// TIA Portal project "Micromaster4_with_S7_1200" (V14)

(* hardware
DEVICE "S7-1200 station_1"  S7-1200 Station
   slot 0: "Rack_0"  S7-1200 Rack  Rack  V1.0
   slot 1: "PLC_1"  CPU 1214C DC/DC/DC  6ES7 214-1AE30-0XB0  V2.0
   slot 2: "AI 4x13BIT_1"  SM 1231 AI4  6ES7 231-4HD30-0XB0  V1.0
   slot 3: "AI 4x13BIT_2"  SM 1231 AI4  6ES7 231-4HD30-0XB0  V1.0
   slot 4: "AQ 2x14BIT_1"  6ES7 232-4HB30-0XB0  V1.0
   slot 101: "CM 1243-5"  CM 1243-5  6GK7 243-5DX30-0XE0  V1.0
DEVICE "GSD device_1"  GSD.Device
   slot 0: "Rack_0"  Rail
   slot 0: "Slave_1"  6SE640X-1PB00-0AA0  V1.0
*)

// ===== PLC "PLC_1"  CPU 1214C DC/DC/DC =====

VAR_GLOBAL   // PLC tag table "Default tag table"
   "Tag_1" AT %M0.0 : Bool;
   "Ready_mode" AT %M0.1 : Bool;
   "Run" AT %M0.2 : Bool;
   "CCW" AT %M0.3 : Bool;
   "OFF2" AT %M0.4 : Bool;
   "OFF3" AT %M0.5 : Bool;
   "Ack" AT %M0.6 : Bool;
   "Control_wrd_1" AT %MW2 : Word;
   "freq" AT %MD4 : Real;
   "write_comm_err" AT %M0.7 : Bool;
   "write_Drive_err" AT %M1.0 : Bool;
   "sent_Dn_flag" AT %M1.1 : Bool;
   "status_wrd" AT %MW8 : Word;
   "actual_freq" AT %MD10 : Real;
   "receive_comm_err" AT %M1.2 : Bool;
   "recieve_dn_flag" AT %M1.3 : Bool;
   "ready_for_on_status" AT %M1.4 : Bool;
   "ready_for_run_status" AT %M1.5 : Bool;
   "operation_on_status" AT %M1.6 : Bool;
   "fault_on" AT %M1.7 : Bool;
   "starting_LOckout__status" AT %M14.0 : Bool;
   "alarm_on" AT %M14.1 : Bool;
   "Motor_overload" AT %M14.2 : Bool;
   "Drive_overload" AT %M14.3 : Bool;
   "Tag_2" AT %MW50 : Word;
   "dummy_bit" AT %M400.1 : Bool;
   "dummy1" AT %MW400 : Word;
   "dummy2" AT %MW402 : Word;
END_VAR

FUNCTION "Micormaster_Write_Data" : Void   // FC1, FBD
TITLE = Micromaster Data Write
{ S7_Optimized_Access := 'TRUE' }
VERSION : 0.1
// Description: This function is used to send the 2 PZD words.
// Author: Ahmed Abd Alrahiem
// Email: a.abdalrahiem@gmail.com
// Last Modification Date: July 9, 2021
   VAR_INPUT
      Control_Word : Word;   // Contains the control word1 that should be transferred to the drive
      Set_Point : Real;   // The set point to be transferred to drive
      WR_HW_ID : Hw_Io;   // The module ID for the PZD words
      Reference_frequency_P2000 : Int;   // The reference frequemcy written to the P2000 parameter
   END_VAR
   VAR_OUTPUT
      Access_Comm_Error : Bool;   // IF set, there is a problem regarding the connection with the drive
      Drive_Error : Bool;   // IF set, there is a problem in the drive and the drive can send no data
      Done : Bool;   // IF set, there is no problem and the data is already written
   END_VAR
   VAR_TEMP
      To_Inverter : Array[1..2] of Word;
      Normalized_setpoint : Word;
      temp_SP_1 : Real;
      temp_SP_2 : Real;
      error_word : Int;
   END_VAR
BEGIN

REGION Network 1
   // Normalization of the setpoint
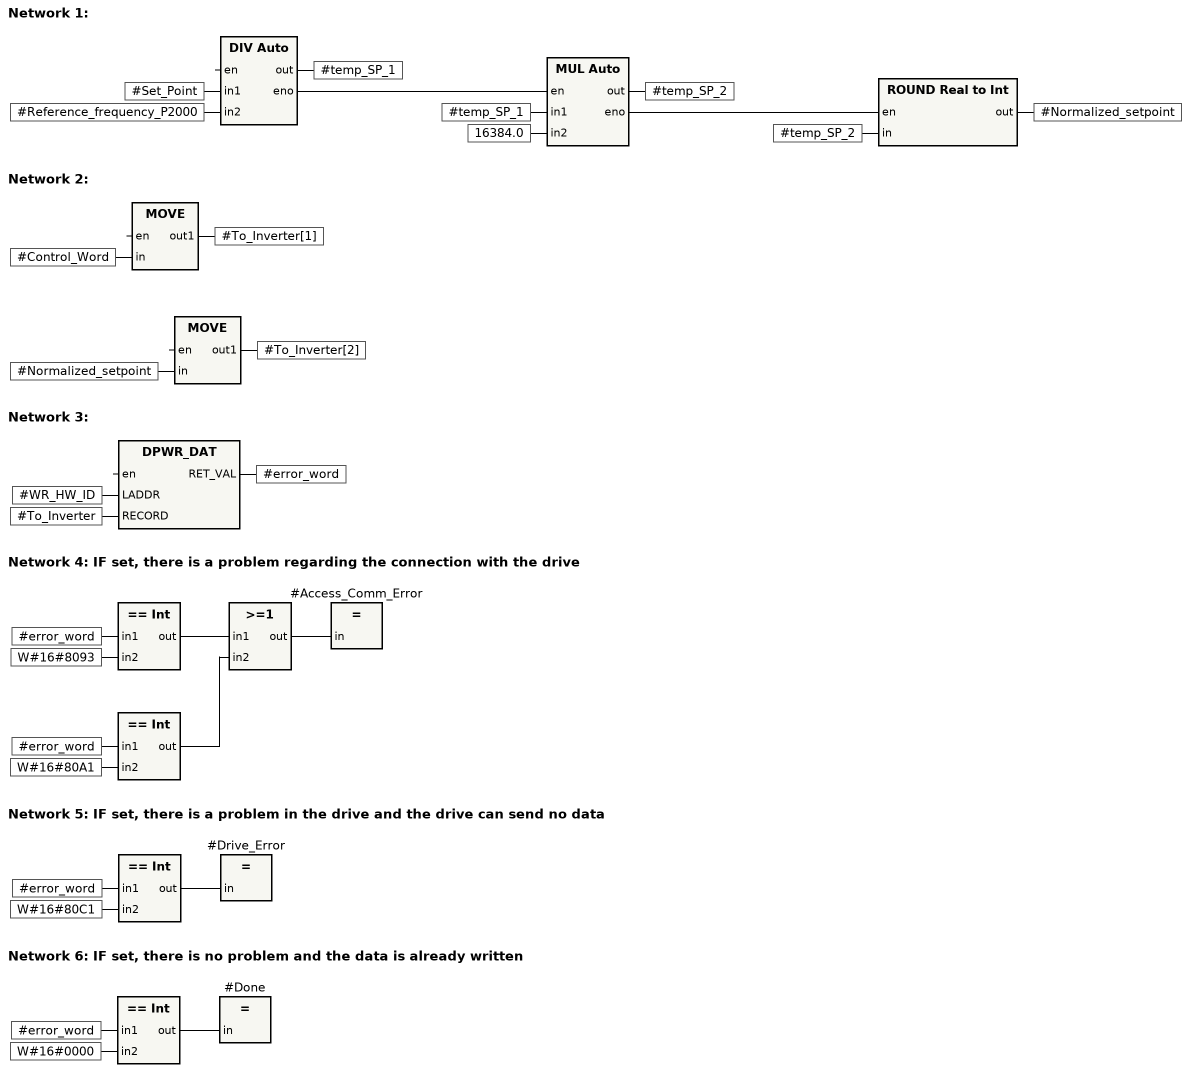
   // ENO of a box is taken as its EN; it also drops when the box reports an error
   #temp_SP_1 := #Set_Point / #Reference_frequency_P2000;
   #temp_SP_2 := #temp_SP_1 * 16384.0;
   #Normalized_setpoint := ROUND(#temp_SP_2);
END_REGION

REGION Network 2
   // This line moves the telegram's control word and setpoint to the same address #To_Inverter
   #To_Inverter[1] := #Control_Word;
   #To_Inverter[2] := #Normalized_setpoint;
END_REGION

REGION Network 3
   // This line writes the data consistently to the inverter
   #error_word := DPWR_DAT(LADDR := #WR_HW_ID, RECORD := #To_Inverter);
END_REGION

REGION Network 4: IF set, there is a problem regarding the connection with the drive
   // The output #Access_Comm_Error is set if there is a problem regarding the connection with the drive
   #Access_Comm_Error := (#error_word = W#16#8093) OR (#error_word = W#16#80A1);
END_REGION

REGION Network 5: IF set, there is a problem in the drive and the drive can send no data
   // The output #Drive_Error is set if there is a problem in the drive and the drive can send no data
   #Drive_Error := #error_word = W#16#80C1;
END_REGION

REGION Network 6: IF set, there is no problem and the data is already written
   // The output #Done is set if there is no problem and the data is already written.
   #Done := #error_word = W#16#0000;
END_REGION
END_FUNCTION

FUNCTION "Micromaster_Control_word1_Generator" : Void   // FC2, FBD
TITLE = Micromaster Control word1 Generator
{ S7_Optimized_Access := 'TRUE' }
VERSION : 0.1
// Description: This function is used to generate the control word to be sent to the Micromaster drive
// Author: Ahmed Abd Alrahiem
// Email: a.abdalrahiem@gmail.com
// Last Modification Date: July 9, 2021
   VAR_INPUT
      "Ready/OFF1" : Bool;   // If set, the inverter will be put in the ready mode--> (bit 0 is set).
      Run : Bool;   // If set, the inverter will be put in the closed loop run mode--> (bit 3 is set).
      CCW_Direction : Bool;   // If set, the motor will run in counter clockwise direction--> (bit 11 is set).
      OFF2 : Bool;   // If set, the drive will coasts to a standstill (Instantaneous braking)-->(bit 1 is reset).
      OFF3 : Bool;   // If set, the drive will shutdown the motor at the fastest possible acceleration rate (rapid shutdown)->(bit 2 is reset).
      Acknowledge_Fault : Bool;   // If set, the inverter fault will be acknowledget--> (bit 7 is set).
   END_VAR
   VAR_OUTPUT
      Control_Word : Word;   // Contains the control word1 that should be transferred to the drive
   END_VAR
   VAR_TEMP
      Control_word_temp1 : Word;
      Control_word_temp2 : Word;
      Control_word_temp3 : Word;
      Control_word_temp4 : Word;
      Control_word_temp5 : Word;
      Control_word_temp6 : Word;
      Control_word_temp7 : Word;
      OFF2_is_reset : Bool;
      OFF3_is_reset : Bool;
   END_VAR
BEGIN

REGION Network 1
   // Moving an initail value equals zero to all bits
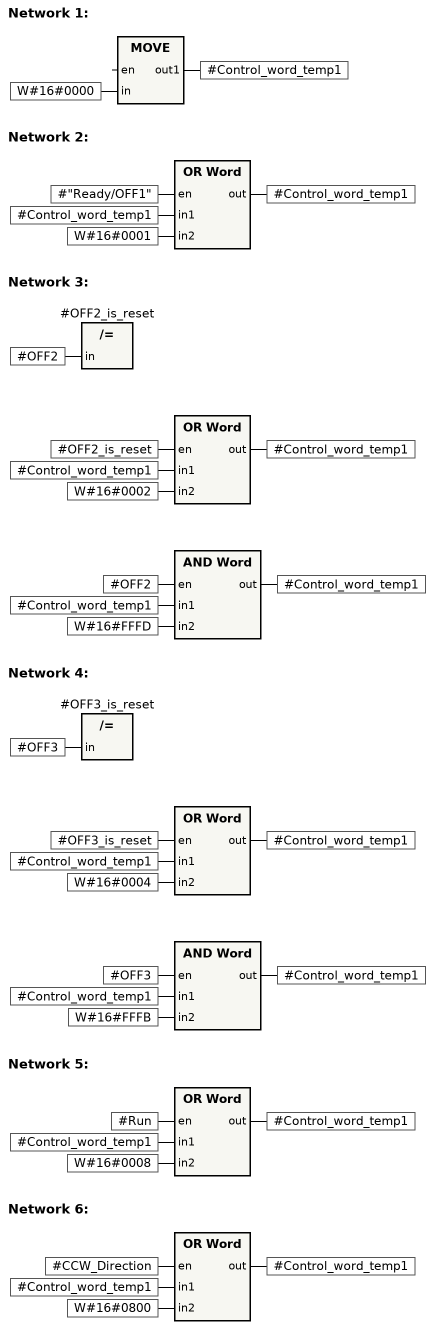
   #Control_word_temp1 := W#16#0000;
END_REGION

REGION Network 2
   // - If the #Ready/OFF1 bit is set, the inverter will be put in the ready mode--> (bit 0 is set).
   // - If the #Ready/OFF1 bit is reset while motor is running, the motor will be brake with ramp time specified in P1121 , deceleration along RFG ramp, pulse disable when f<fmin
   // no checked SCL form for this network; see the picture
END_REGION

REGION Network 3
   // - If the #OFF2 bit is set, the drive will coasts to a standstill (Instantaneous braking)-->(bit 1 is reset).
   // no checked SCL form for this network; see the picture
END_REGION

REGION Network 4
   // - If the #OFF3 bit is set, the drive will shutdown the motor at the fastest possible acceleration rate (rapid shutdown)->(bit 2 is reset).
   // no checked SCL form for this network; see the picture
END_REGION

REGION Network 5
   // - If the #Run bit is set, the inverter will be put in the closed loop run mode--> (bit 3 is set).
   // no checked SCL form for this network; see the picture
END_REGION

REGION Network 6
   // - If the #CCW_Direction bit is set, the motor will run in counter clockwise direction--> (bit 11 is set).
   // no checked SCL form for this network; see the picture
END_REGION

REGION Network 7
   // - If the #Acknowledge_Fault bit is set, the inverter fault will be acknowledget--> (bit 7 is set).
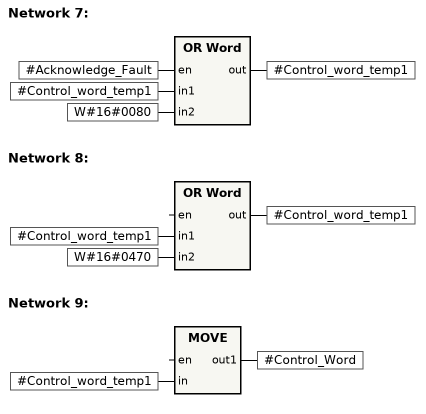
   // no checked SCL form for this network; see the picture
END_REGION

REGION Network 8
   // no checked SCL form for this network; see the picture
END_REGION

REGION Network 9
   #Control_Word := #Control_word_temp1;
END_REGION
END_FUNCTION

FUNCTION "Micromaster_Status_Word1_Reader" : Void   // FC3, FBD
TITLE = Micromaster Control word1 Reader
{ S7_Optimized_Access := 'TRUE' }
VERSION : 0.1
// Description: This function is used to interpret the status word recieved the Micromaster drive
// Author: Ahmed Abd Alrahiem
// Email: a.abdalrahiem@gmail.com
// Last Modification Date: July 9, 2021
   VAR_INPUT
      Status_Word : Word;   // This is the status word 1 recieved from the drive
   END_VAR
   VAR_OUTPUT
      Ready_for_ON : Bool;   // If set, means Power supply switched on, electronics initialized, pulses disabled
      Ready_to_Run : Bool;   // If set, Converter is switched on (ON command is applied), no fault is active, inverter can start when "Enable operation" command is ssued.
      Operation_is_Enabled : Bool;   // If set, Operation is enabled
      Fault_is_Active : Bool;   // If set, Drive is faulty and thus inoperative, switches to starting lockout state after successful correction and acknowledgement of fault.
      Starting_Lockout : Bool;   // If set, Drive can be restarted only by OFF1 followed by ON
      Alarm_is_Active : Bool;   // If set, there is a warning but drive still in operation.
      Motor_Overload : Bool;   // If set, Motor data indicate overload condition
      Drive_Overload : Bool;   // If set, converter is in overload condition(eg:current or temperature)
   END_VAR
   VAR_TEMP
      temp1 : Word;
      temp2 : Word;
      temp3 : Word;
      temp4 : Word;
      temp5 : Word;
      temp6 : Word;
      temp7 : Word;
      temp8 : Word;
      temp9 : Word;
   END_VAR
BEGIN

REGION Network 1: If set, means Power supply switched on, electronics initialized, pulses disabled
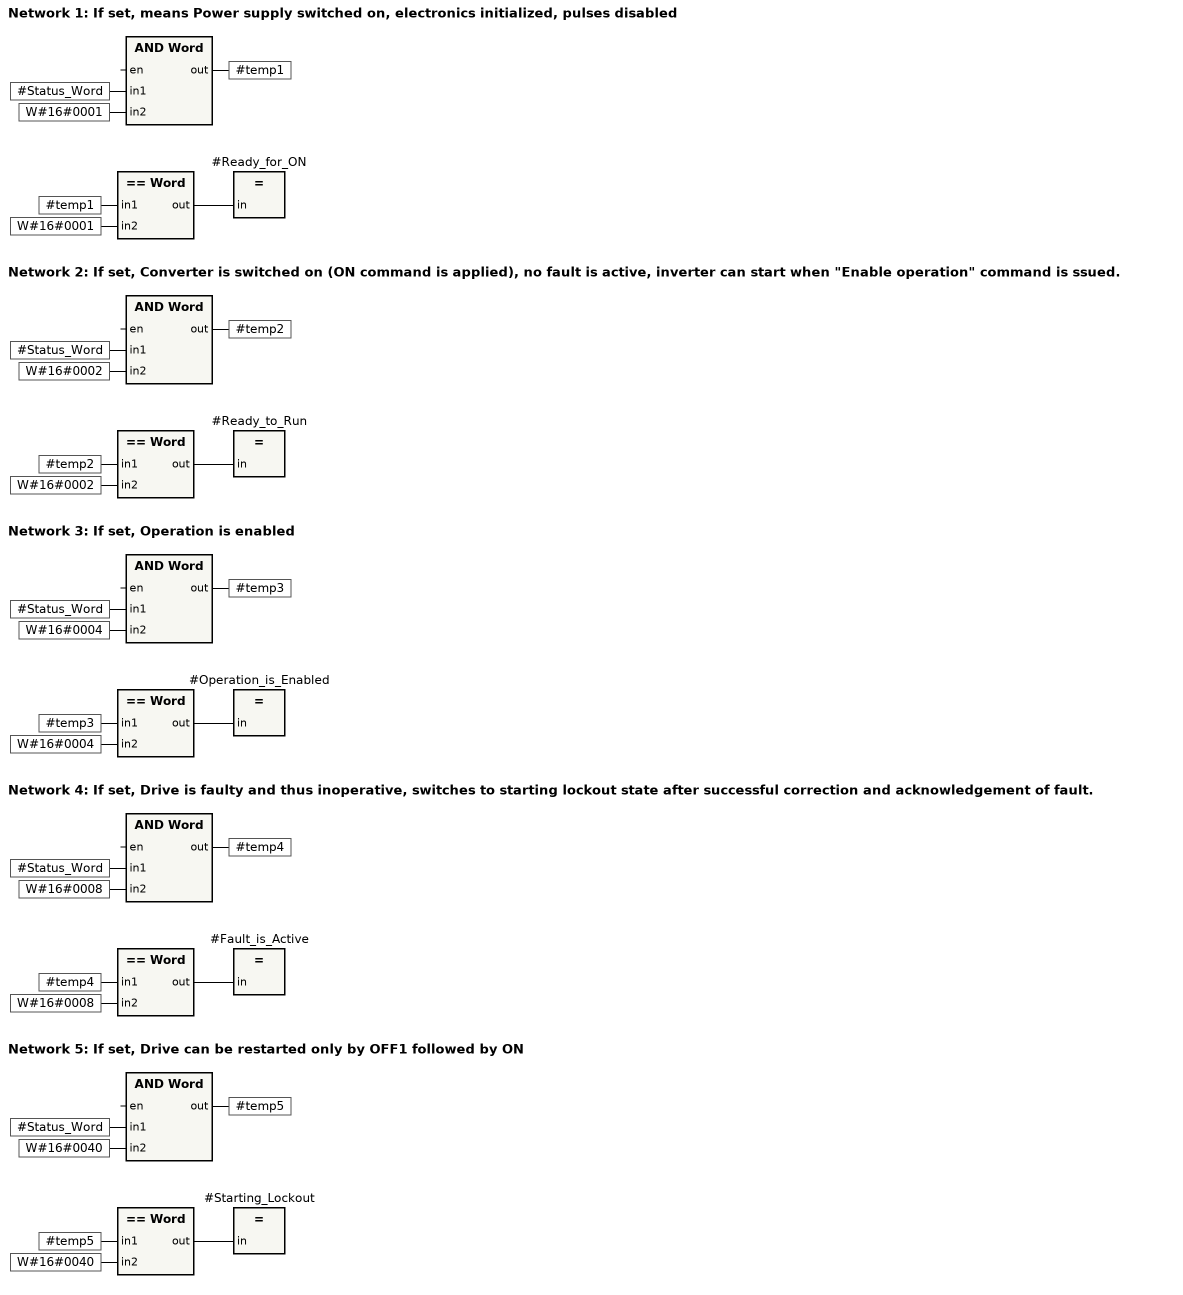
   // no checked SCL form for this network; see the picture
END_REGION

REGION Network 2: If set, Converter is switched on (ON command is applied), no fault is active, inverter can start when "Enable operation" command is ssued.
   // no checked SCL form for this network; see the picture
END_REGION

REGION Network 3: If set, Operation is enabled
   // no checked SCL form for this network; see the picture
END_REGION

REGION Network 4: If set, Drive is faulty and thus inoperative, switches to starting lockout state after successful correction and acknowledgement of fault.
   // no checked SCL form for this network; see the picture
END_REGION

REGION Network 5: If set, Drive can be restarted only by OFF1 followed by ON
   // no checked SCL form for this network; see the picture
END_REGION

REGION Network 6: If set, there is a warning but drive still in operation.
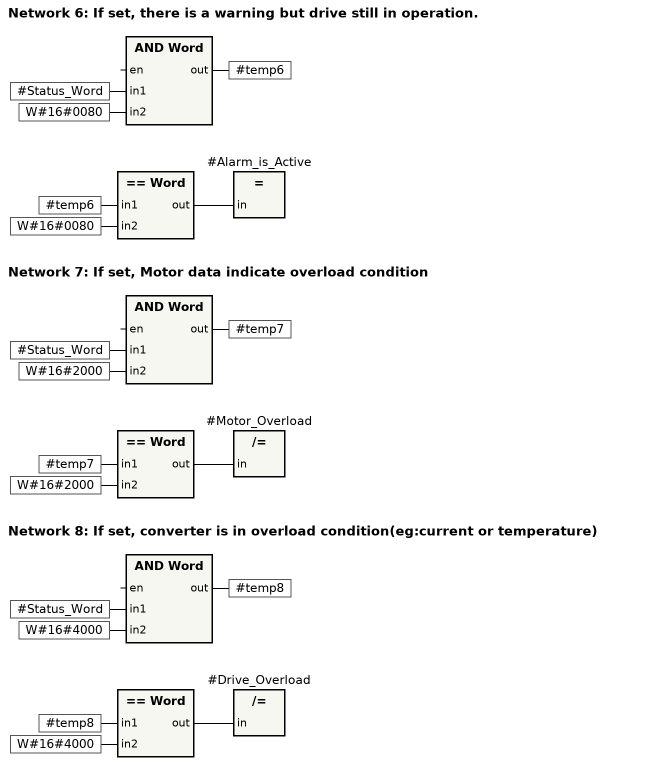
   // no checked SCL form for this network; see the picture
END_REGION

REGION Network 7: If set, Motor data indicate overload condition
   // no checked SCL form for this network; see the picture
END_REGION

REGION Network 8: If set, converter is in overload condition(eg:current or temperature)
   // no checked SCL form for this network; see the picture
END_REGION
END_FUNCTION

FUNCTION "Micormaster_read_Data" : Void   // FC4, FBD
TITLE = Micromaster Data Read
{ S7_Optimized_Access := 'TRUE' }
VERSION : 0.1
// Description: This function is used to recieve the status word and the actual speed from the Micromaster drive.
// Author: Ahmed Abd Alrahiem
// Email: a.abdalrahiem@gmail.com
// Last Modification Date: July 9, 2021
   VAR_INPUT
      RD_HW_ID : Hw_Io;   // The module ID for the PZD words
      Reference_frequency_P2000 : Int;   // The reference frequemcy written to the P2000 parameter
   END_VAR
   VAR_OUTPUT
      Status_Word : Word;   // The status word 1 recieved from the drive
      Actual_Speed : Real;   // The actual frequency recieved from the drive
      Access_Comm_Error : Bool;   // IF set, there is a problem regarding the connection with the drive
      Done : Bool;   // IF set, there is no problem and the data is already read.
   END_VAR
   VAR_TEMP
      from_Inverter : Array[1..2] of Word;
      Denormalized_setpoint : Real;
      temp_SP_1 : Real;
      temp_SP_2 : Real;
      error_word : Int;
   END_VAR
BEGIN

REGION Network 1
   // Reading the data consistently from the drive with the hardware_id = #RD_HW_ID
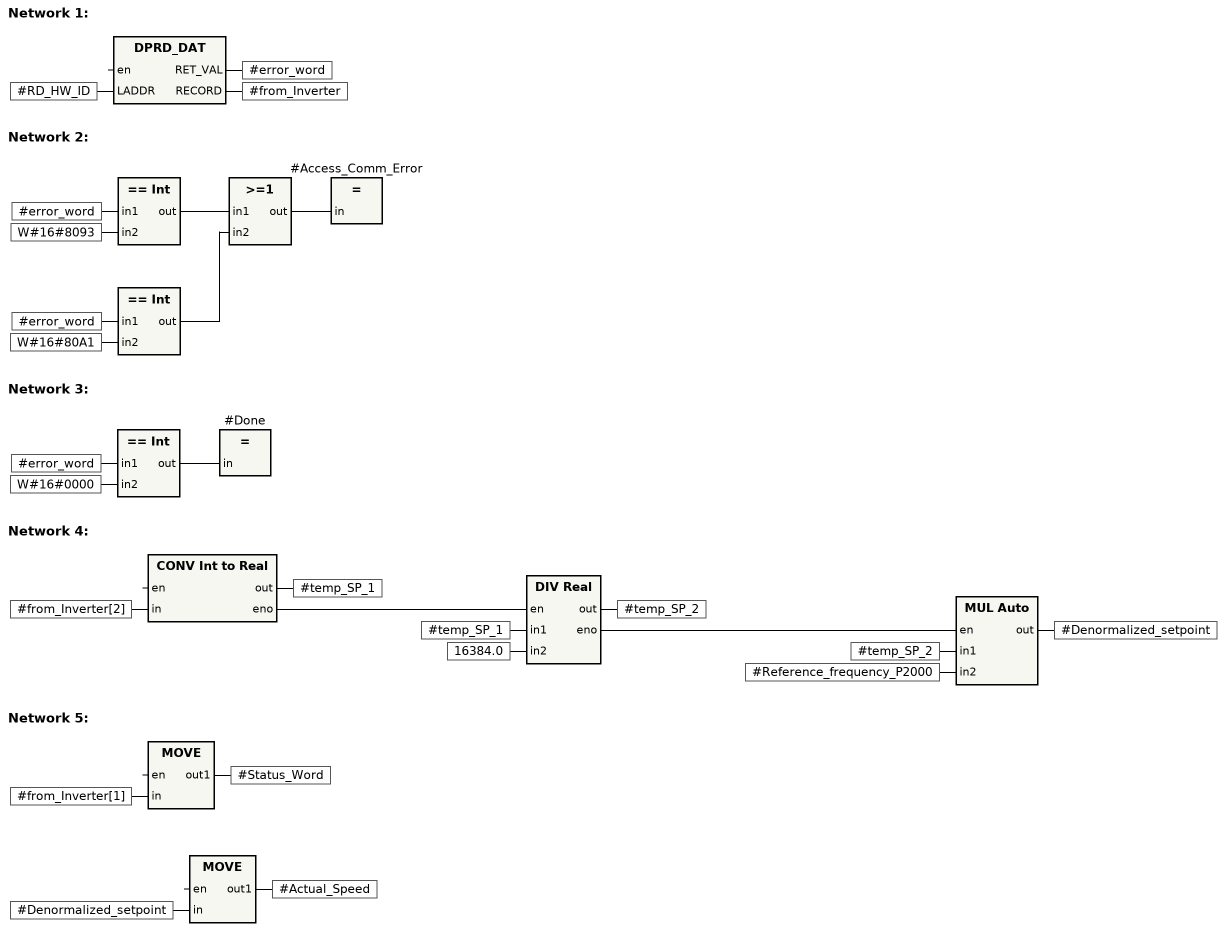
   #error_word := DPRD_DAT(LADDR := #RD_HW_ID, RECORD => #from_Inverter);
END_REGION

REGION Network 2
   // The output #Access_Comm_Error is set if there is a problem regarding the connection with the drive
   #Access_Comm_Error := (#error_word = W#16#8093) OR (#error_word = W#16#80A1);
END_REGION

REGION Network 3
   // The output #Done is set if there is no problem and the data is already read.
   #Done := #error_word = W#16#0000;
END_REGION

REGION Network 4
   // Denormalization of the actual spead
   // ENO of a box is taken as its EN; it also drops when the box reports an error
   #temp_SP_1 := INT_TO_REAL(#from_Inverter[2]);
   #temp_SP_2 := #temp_SP_1 / 16384.0;
   #Denormalized_setpoint := #temp_SP_2 * #Reference_frequency_P2000;
END_REGION

REGION Network 5
   // This line outputs the status word and the actual speed
   #Status_Word := #from_Inverter[1];
   #Actual_Speed := #Denormalized_setpoint;
END_REGION
END_FUNCTION

ORGANIZATION_BLOCK "Main"   // OB1, FBD, ProgramCycle
TITLE = "Main Program Sweep (Cycle)"
{ S7_Optimized_Access := 'TRUE' }
VERSION : 0.1
BEGIN

REGION Network 1
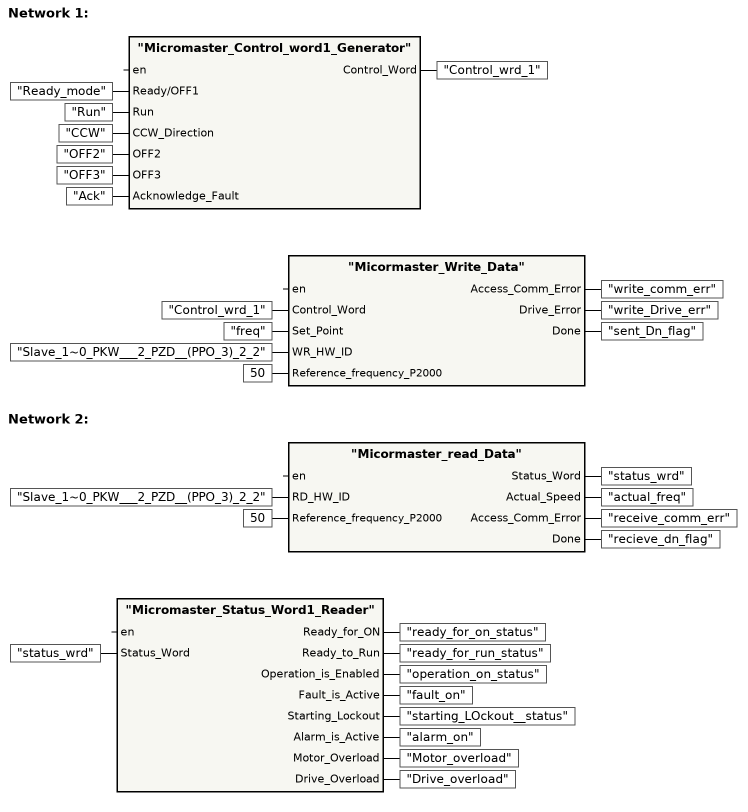
   "Micromaster_Control_word1_Generator"("Ready/OFF1" := "Ready_mode",
                           Run := "Run",
                           CCW_Direction := "CCW",
                           OFF2 := "OFF2",
                           OFF3 := "OFF3",
                           Acknowledge_Fault := "Ack",
                           Control_Word => "Control_wrd_1");
   "Micormaster_Write_Data"(Control_Word := "Control_wrd_1",
                           Set_Point := "freq",
                           WR_HW_ID := "Slave_1~0_PKW___2_PZD__(PPO_3)_2_2",
                           Reference_frequency_P2000 := 50,
                           Access_Comm_Error => "write_comm_err",
                           Drive_Error => "write_Drive_err",
                           Done => "sent_Dn_flag");
END_REGION

REGION Network 2
   "Micormaster_read_Data"(RD_HW_ID := "Slave_1~0_PKW___2_PZD__(PPO_3)_2_2",
                           Reference_frequency_P2000 := 50,
                           Status_Word => "status_wrd",
                           Actual_Speed => "actual_freq",
                           Access_Comm_Error => "receive_comm_err",
                           Done => "recieve_dn_flag");
   "Micromaster_Status_Word1_Reader"(Status_Word := "status_wrd",
                           Ready_for_ON => "ready_for_on_status",
                           Ready_to_Run => "ready_for_run_status",
                           Operation_is_Enabled => "operation_on_status",
                           Fault_is_Active => "fault_on",
                           Starting_Lockout => "starting_LOckout__status",
                           Alarm_is_Active => "alarm_on",
                           Motor_Overload => "Motor_overload",
                           Drive_Overload => "Drive_overload");
END_REGION
END_ORGANIZATION_BLOCK